// TIA Portal V20 export
FUNCTION "MoveAny256" : Void   // FC100, LAD
TITLE = Move ANY 256
VERSION : 1.0
// Copy any data type - max length 256 bytes
// stored: IsIECCheckEnabled true, Namespace CITI_Logic, SetENOAutomatically false
   VAR_INPUT
      iSource : Variant;
   END_VAR
   VAR_OUTPUT
      iTarget : Variant;
   END_VAR
   VAR_TEMP
      tempClearByte : Byte;
      tempRetVal : Int;
      tempPos : DInt;
      tempStore : Array[0..999] of Byte;
   END_VAR
BEGIN

REGION Network 1
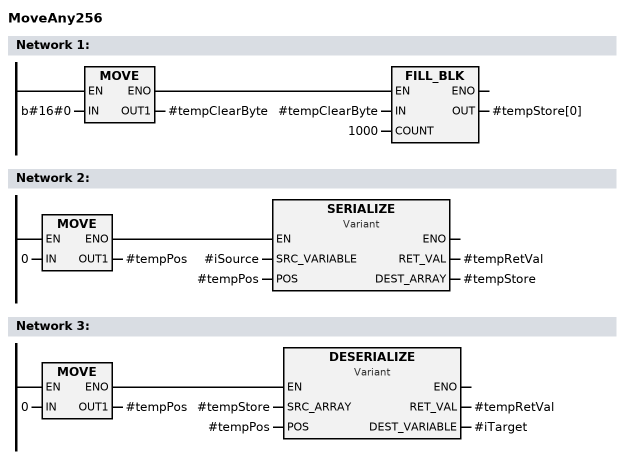
   RUNG wire#powerrail
      Move(in := b#16#0, out1 => #tempClearByte)
      FillBlockI(in := #tempClearByte, count := 1000, out => #tempStore[0])
   END_RUNG
   // the same network as SCL:
   #tempClearByte := b#16#0;
   FILL_BLK(IN := #tempClearByte, COUNT := 1000, OUT => #tempStore[0]);
END_REGION

REGION Network 2
   RUNG wire#powerrail
      Move(in := 0, out1 => #tempPos)
      { S7_Templates := "[src_type := Variant, dest_type := Variant]" } Serialize(SRC_VARIABLE := #iSource, POS := #tempPos, Ret_Val => #tempRetVal, DEST_ARRAY => #tempStore)
   END_RUNG
   // the same network as SCL:
   #tempPos := 0;
   #tempRetVal := Serialize(SRC_VARIABLE := #iSource, POS := #tempPos, DEST_ARRAY => #tempStore);
END_REGION

REGION Network 3
   RUNG wire#powerrail
      Move(in := 0, out1 => #tempPos)
      { S7_Templates := "[src_type := Variant, dest_type := Variant]" } Deserialize(SRC_ARRAY := #tempStore, POS := #tempPos, Ret_Val => #tempRetVal, DEST_VARIABLE => #iTarget)
   END_RUNG
   // the same network as SCL:
   #tempPos := 0;
   #tempRetVal := Deserialize(SRC_ARRAY := #tempStore, POS := #tempPos, DEST_VARIABLE => #iTarget);
END_REGION
END_FUNCTION
